{attribute 'linkalways'}
{attribute 'hide_all_locals'}
FUNCTION_BLOCK ValueDate EXTENDS ValueDateRead IMPLEMENTS Value
VAR
END_VAR

METHOD SetFromType : BOOL
VAR_INPUT
	source : __SYSTEM.AnyType;
END_VAR
SetFromType := ConvertAnyType(source, thisAnyType);
END_METHOD

METHOD SetFromString : BOOL
VAR_INPUT
	value : T_MaxString;
END_VAR
thisValue := STRING_TO_DATE(value);

SetFromString := TRUE;
END_METHOD

METHOD Set : BOOL
VAR_INPUT
	source : ANY;
END_VAR
Set := ConvertAnyType(source, thisAnyType);
END_METHOD

END_FUNCTION_BLOCK

(* stored: Version 1.1.0.1
   POU ValueDate: Id {5a79daf1-1dac-48b5-b4a6-b0903b6f3c21}, SpecialFunc None
   Method SetFromType: Id {9aab414d-4da0-4969-b17c-6b51b1d1e1df}
   Method SetFromString: Id {dec82281-028e-43c0-ad37-fb97cce09eef}
   Method Set: Id {553662da-a971-44ca-ad65-9e3ffe3c9772} *)
